// Latched by the base on the Execute rising edge (S6.1).
TYPE ST_SeparatorParCmd :
STRUCT
    OpenStopper : BOOL;   // OPEN_CLOSE: TRUE = open, FALSE = close
END_STRUCT
END_TYPE

(* stored: Version 1.1.0.1, ProductVersion 3.1.4024.12
   DUT ST_SeparatorParCmd: Id {90674489-497d-4a1e-9bc3-77e1ed34ecf1} *)
